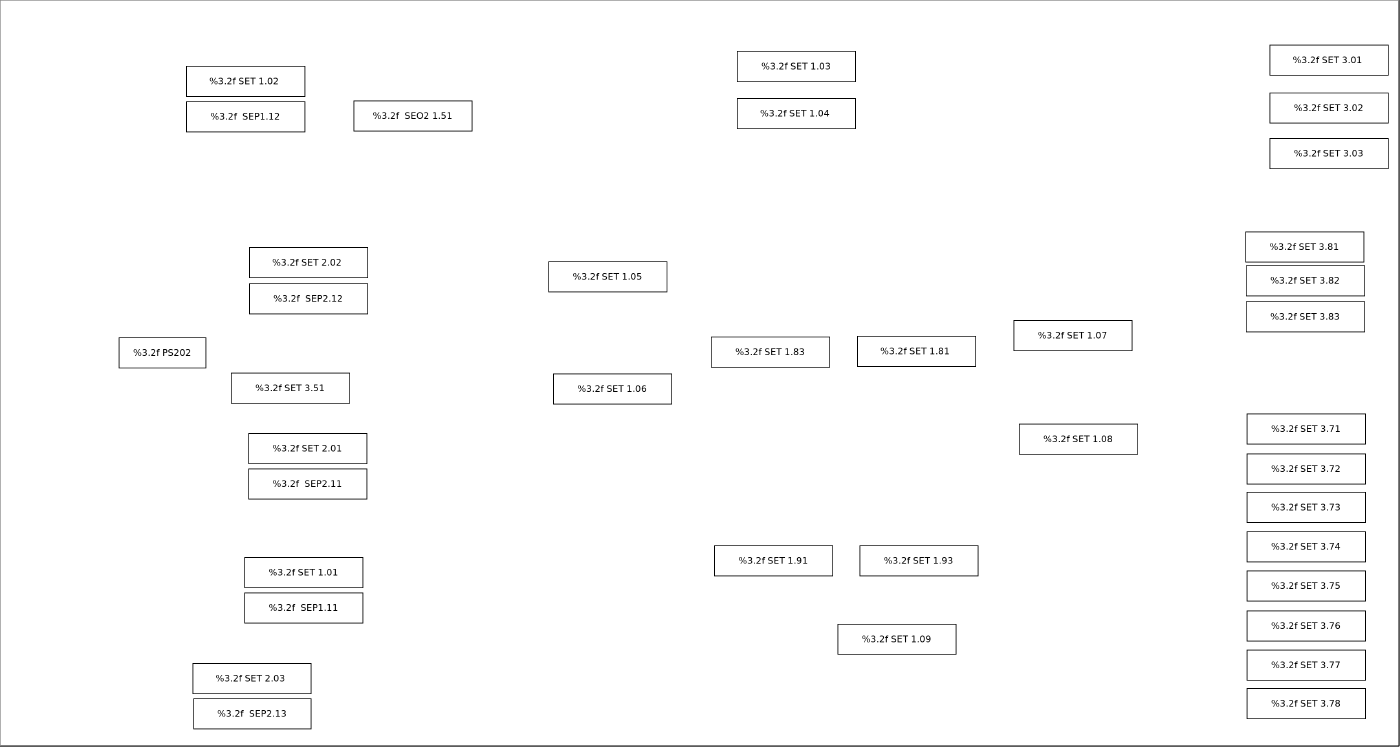
VISUALIZATION Layout  // 1782x952, background image LAyout
    Rectangle (0,950 1780x2)
    Rectangle (1780,0 2x950)
    Rectangle (311,710 151x39), "%3.2f SET 1.01", tooltip "Durchmesser in mm eingeben", text variable: GVL.T_Vor_WT_Visu
    Rectangle (237,84 151x39), "%3.2f SET 1.02", tooltip "Durchmesser in mm eingeben", text variable: GVL.T_nach_WT_Visu
    Rectangle (237,129 151x39), "%3.2f SEP1.12", tooltip "Durchmesser in mm eingeben", text variable: P_nach_WT_Visu
    Rectangle (450,128 151x39), "%3.2f SEO2 1.51", tooltip "Durchmesser in mm eingeben", text variable: GVL.O2_Visu
    Rectangle (317,315 151x39), "%3.2f SET 2.02", tooltip "Durchmesser in mm eingeben", text variable: GVL.T_Komp_Auslass_Visu
    Rectangle (317,361 151x39), "%3.2f SEP2.12", tooltip "Durchmesser in mm eingeben", text variable: GVL.P_Komp_Auslass_Visu
    Rectangle (316,597 151x39), "%3.2f SEP2.11", tooltip "Durchmesser in mm eingeben", text variable: GVL.P_Komp_Einlass_Visu
    Rectangle (294,475 151x39), "%3.2f SET 3.51", tooltip "Durchmesser in mm eingeben", text variable: GVL.T_DK_Steigband3_Visu
    Rectangle (316,552 151x39), "%3.2f SET 2.01", tooltip "Durchmesser in mm eingeben", text variable: GVL.T_Komp_Einlass_Visu
    Rectangle (245,845 151x39), "%3.2f SET 2.03", tooltip "Durchmesser in mm eingeben", text variable: GVL.T_Kond_Auslass_Visu
    Rectangle (311,755 151x39), "%3.2f SEP1.11", tooltip "Durchmesser in mm eingeben", text variable: GVL.P_Vor_WT_Visu
    Rectangle (698,333 151x39), "%3.2f SET 1.05", tooltip "Durchmesser in mm eingeben", text variable: GVL.T_Einduesung_Oben_Visu
    Rectangle (704,476 151x39), "%3.2f SET 1.06", tooltip "Durchmesser in mm eingeben", text variable: GVL.T_Einduesung_Unten_Visu
    Rectangle (938,65 151x39), "%3.2f SET 1.03", tooltip "Durchmesser in mm eingeben", text variable: T_HE_Einduesung_Oben_Visu
    Rectangle (938,125 151x39), "%3.2f SET 1.04", tooltip "Durchmesser in mm eingeben", text variable: T_HE_Einduesung_Unten_Visu
    Rectangle (905,429 151x39), "%3.2f SET 1.83", tooltip "Durchmesser in mm eingeben", text variable: GVL.T_DK_Band_oben3_Visu
    Rectangle (1091,428 151x39), "%3.2f SET 1.81", tooltip "Durchmesser in mm eingeben", text variable: GVL.T_DK_Band_oben1_Visu
    Rectangle (909,695 151x39), "%3.2f SET 1.91", tooltip "Durchmesser in mm eingeben", text variable: GVL.T_DK_Band_unten1_Visu
    Rectangle (1094,695 151x39), "%3.2f SET 1.93", tooltip "Durchmesser in mm eingeben", text variable: GVL.T_DK_Band_unten3_Visu
    Rectangle (1290,408 151x39), "%3.2f SET 1.07", tooltip "Durchmesser in mm eingeben", text variable: GVL.T_Absaugung_Oben_Visu
    Rectangle (1297,540 151x39), "%3.2f SET 1.08", tooltip "Durchmesser in mm eingeben", text variable: GVL.T_Absaugung_Unten_Visu
    Rectangle (1066,795 151x39), "%3.2f SET 1.09", tooltip "Durchmesser in mm eingeben", text variable: GVL.T_Vor_UmdampfLuefter_Visu
    Rectangle (1616,57 151x39), "%3.2f SET 3.01", tooltip "Durchmesser in mm eingeben", text variable: GVL.T_DK_Oben_Visu
    Rectangle (1616,118 151x39), "%3.2f SET 3.02", tooltip "Durchmesser in mm eingeben", text variable: GVL.T_DK_Mitte_Visu
    Rectangle (1616,176 151x39), "%3.2f SET 3.03", tooltip "Durchmesser in mm eingeben", text variable: GVL.T_DK_Unten_Visu
    Rectangle (1587,527 151x39), "%3.2f SET 3.71", tooltip "Durchmesser in mm eingeben", text variable: GVL.T_Mat_Auslass1_Visu
    Rectangle (1587,578 151x39), "%3.2f SET 3.72", tooltip "Durchmesser in mm eingeben", text variable: GVL.T_Mat_Auslass2_Visu
    Rectangle (1587,627 151x39), "%3.2f SET 3.73", tooltip "Durchmesser in mm eingeben", text variable: GVL.T_Mat_Auslass3_Visu
    Rectangle (1587,677 151x39), "%3.2f SET 3.74", tooltip "Durchmesser in mm eingeben", text variable: GVL.T_Mat_Auslass4_Visu
    Rectangle (1587,727 151x39), "%3.2f SET 3.75", tooltip "Durchmesser in mm eingeben", text variable: GVL.T_Mat_Auslass5_Visu
    Rectangle (1587,778 151x39), "%3.2f SET 3.76", tooltip "Durchmesser in mm eingeben", text variable: GVL.T_Mat_Auslass6_Visu
    Rectangle (1587,828 151x39), "%3.2f SET 3.77", tooltip "Durchmesser in mm eingeben", text variable: GVL.T_Mat_Auslass7_Visu
    Rectangle (1587,877 151x39), "%3.2f SET 3.78", tooltip "Durchmesser in mm eingeben", text variable: GVL.T_Mat_Auslass8_Visu
    Rectangle (1585,295 151x39), "%3.2f SET 3.81", tooltip "Durchmesser in mm eingeben", text variable: GVL.T_DK_Steigband1_Visu
    Rectangle (1586,338 151x39), "%3.2f SET 3.82", tooltip "Durchmesser in mm eingeben", text variable: GVL.T_DK_Steigband2_Visu
    Rectangle (1586,384 151x39), "%3.2f SET 3.83", tooltip "Durchmesser in mm eingeben", text variable: GVL.T_DK_Steigband3_Visu
    Rectangle (246,890 150x39), "%3.2f SEP2.13", tooltip "Durchmesser in mm eingeben", text variable: GVL.P_Kond_Auslass_Visu
    Rectangle (151,430 111x39), "%3.2f PS202", tooltip "Durchmesser in mm eingeben", text variable: Ps_202
END_VISUALIZATION

(* stored: Version 1.1.0.1, ProductVersion 3.1.4024.3
   Visu Layout: Id {7e7cc8d6-7487-48f0-9b06-23c59805f660} *)
